   A_3126_TSC01_AC.Msg.WarningDoneL := FALSE;
   A_3126_TSC01_AC.Msg.WarningDoneMid := FALSE;
   A_3126_TSC01_AC.Msg.WarningDoneH := FALSE;
   A_3126_TSC01_AC.Msg.WarningDoneHH := FALSE;
   A_3126_TSC01_AC.Msg.FaultDoneLL := FALSE;
   A_3126_TSC01_AC.Msg.FaultDoneL := FALSE;
   A_3126_TSC01_AC.Msg.FaultDoneMid := FALSE;
   A_3126_TSC01_AC.Msg.FaultDoneH := FALSE;
   A_3126_TSC01_AC.Msg.FaultDoneHH := FALSE;
   A_3126_TSC01_AC.Msg.FaultDoneDev := FALSE;
   A_3126_TSC01_AC.Msg.FaultDoneAI := FALSE;
   A_3126_TSC01_AC.OutAlarmNrLog := 0;
   A_3126_TSC01_AC.Par.ParObjectNo := 27124;
   A_3126_TSC01_AC.Par.ParMsgType := 7252;
   A_3126_TSC01_AC.Par.ParHornCode := 10;
   A_3126_TSC01_AC.Par.ParLogOff := FALSE;
   A_3126_TSC01_AC.Par.ParSpare0401 := FALSE;
   A_3126_TSC01_AC.Par.ParValueByUser := FALSE;
   A_3126_TSC01_AC.Par.ParLimitsPc := TRUE;
   A_3126_TSC01_AC.Par.ParWago := FALSE;
   A_3126_TSC01_AC.Par.ParNoHornByWarning := FALSE;
   A_3126_TSC01_AC.Par.ParWarningLL := FALSE;
   A_3126_TSC01_AC.Par.ParWarningL := FALSE;
   A_3126_TSC01_AC.Par.ParWarningMid := FALSE;
   A_3126_TSC01_AC.Par.ParWarningH := FALSE;
   A_3126_TSC01_AC.Par.ParWarningHH := FALSE;
   A_3126_TSC01_AC.Par.ParPreAlarmLL := FALSE;
   A_3126_TSC01_AC.Par.ParPreAlarmL := FALSE;
   A_3126_TSC01_AC.Par.ParPreAlarmMid := FALSE;
   A_3126_TSC01_AC.Par.ParPreAlarmH := FALSE;
   A_3126_TSC01_AC.Par.ParPreAlarmHH := FALSE;
   A_3126_TSC01_AC.Par.ParUnitsByZeroDigit := L#0;
   A_3126_TSC01_AC.Par.ParUnitsByMaxDigit := L#25384;
   A_3126_TSC01_AC.Par.ParUnitsBy100Pc := L#10000;
   A_3126_TSC01_AC.Par.ParLimitLL := L#-1;
   A_3126_TSC01_AC.Par.ParLimitL := L#0;
   A_3126_TSC01_AC.Par.ParLimitH := L#5400;
   A_3126_TSC01_AC.Par.ParLimitHH := L#6000;
   A_3126_TSC01_AC.Par.ParMonTimeLL := 0;
   A_3126_TSC01_AC.Par.ParMonTimeL := 0;
   A_3126_TSC01_AC.Par.ParMonTimeMid := 0;
   A_3126_TSC01_AC.Par.ParMonTimeH := 0;
   A_3126_TSC01_AC.Par.ParMonTimeHH := 0;
   A_3126_TSC01_AC.Par.ParDelayTimeDown := 10;
   A_3126_TSC01_AC.Par.ParDelayTimeUp := 10;
   A_3126_TSC01_AC.Par.ParDelayTime := 30;
   A_3126_TSC01_AC.Par.OutMonTimeLL := 0;
   A_3126_TSC01_AC.Par.OutMonTimeL := 0;
   A_3126_TSC01_AC.Par.OutMonTimeMid := 0;
   A_3126_TSC01_AC.Par.OutMonTimeH := 0;
   A_3126_TSC01_AC.Par.OutMonTimeHH := 0;
   A_3126_TSC01_AC.Par.OutDelayTimeDown := 0;
   A_3126_TSC01_AC.Par.OutDelayTimeUp := 0;
   A_3126_TSC01_AC.Par.OutDelayTime := 0;
   A_3126_TSC01_AC.Par.Spare66 := 0;
   A_3126_TSC01_AF.StCode := 0;
   A_3126_TSC01_AF.InMonLL := FALSE;
   A_3126_TSC01_AF.InMonL := FALSE;
   A_3126_TSC01_AF.InMonMid := FALSE;
   A_3126_TSC01_AF.InMonH := FALSE;
   A_3126_TSC01_AF.InMonHH := FALSE;
   A_3126_TSC01_AF.spare0205 := FALSE;
   A_3126_TSC01_AF.InpFaultAI := FALSE;
   A_3126_TSC01_AF.InpFaultDev := FALSE;
   A_3126_TSC01_AF.InHWStop := FALSE;
   A_3126_TSC01_AF.InDPFault := FALSE;
   A_3126_TSC01_AF.InDisable := FALSE;
   A_3126_TSC01_AF.CmdFaultReset := FALSE;
   A_3126_TSC01_AF.InLocal := FALSE;
   A_3126_TSC01_AF.spare0305 := FALSE;
   A_3126_TSC01_AF.InReport := FALSE;
   A_3126_TSC01_AF.spare0307 := FALSE;
   A_3126_TSC01_AF.OutLL := FALSE;
   A_3126_TSC01_AF.OutL := FALSE;
   A_3126_TSC01_AF.OutH := FALSE;
   A_3126_TSC01_AF.OutHH := FALSE;
   A_3126_TSC01_AF.OutOverflow := FALSE;
   A_3126_TSC01_AF.spare0405 := FALSE;
   A_3126_TSC01_AF.OutFaultAI := FALSE;
   A_3126_TSC01_AF.spare0407 := FALSE;
   A_3126_TSC01_AF.StLL := FALSE;
   A_3126_TSC01_AF.StL := FALSE;
   A_3126_TSC01_AF.StMid := FALSE;
   A_3126_TSC01_AF.StH := FALSE;
   A_3126_TSC01_AF.StHH := FALSE;
   A_3126_TSC01_AF.StFaultAI := FALSE;
   A_3126_TSC01_AF.OutWarning := FALSE;
   A_3126_TSC01_AF.OutFaulted := FALSE;
   A_3126_TSC01_AF.InpValue := 0;
   A_3126_TSC01_AF.OutValuePc := 0;
   A_3126_TSC01_AF.OutValueUnits := L#0;
   A_3126_TSC01_AF.Msg.WarningDoneLL := FALSE;
   A_3126_TSC01_AF.Msg.WarningDoneL := FALSE;
   A_3126_TSC01_AF.Msg.WarningDoneMid := FALSE;
   A_3126_TSC01_AF.Msg.WarningDoneH := FALSE;
   A_3126_TSC01_AF.Msg.WarningDoneHH := FALSE;
   A_3126_TSC01_AF.Msg.FaultDoneLL := FALSE;
   A_3126_TSC01_AF.Msg.FaultDoneL := FALSE;
   A_3126_TSC01_AF.Msg.FaultDoneMid := FALSE;
   A_3126_TSC01_AF.Msg.FaultDoneH := FALSE;
   A_3126_TSC01_AF.Msg.FaultDoneHH := FALSE;
   A_3126_TSC01_AF.Msg.FaultDoneDev := FALSE;
   A_3126_TSC01_AF.Msg.FaultDoneAI := FALSE;
   A_3126_TSC01_AF.OutAlarmNrLog := 0;
   A_3126_TSC01_AF.Par.ParObjectNo := 27125;
   A_3126_TSC01_AF.Par.ParMsgType := 7252;
   A_3126_TSC01_AF.Par.ParHornCode := 10;
   A_3126_TSC01_AF.Par.ParLogOff := FALSE;
   A_3126_TSC01_AF.Par.ParSpare0401 := FALSE;
   A_3126_TSC01_AF.Par.ParValueByUser := FALSE;
   A_3126_TSC01_AF.Par.ParLimitsPc := TRUE;
   A_3126_TSC01_AF.Par.ParWago := FALSE;
   A_3126_TSC01_AF.Par.ParNoHornByWarning := FALSE;
   A_3126_TSC01_AF.Par.ParWarningLL := FALSE;
   A_3126_TSC01_AF.Par.ParWarningL := FALSE;
   A_3126_TSC01_AF.Par.ParWarningMid := FALSE;
   A_3126_TSC01_AF.Par.ParWarningH := FALSE;
   A_3126_TSC01_AF.Par.ParWarningHH := FALSE;
   A_3126_TSC01_AF.Par.ParPreAlarmLL := FALSE;
   A_3126_TSC01_AF.Par.ParPreAlarmL := FALSE;
   A_3126_TSC01_AF.Par.ParPreAlarmMid := FALSE;
   A_3126_TSC01_AF.Par.ParPreAlarmH := FALSE;
   A_3126_TSC01_AF.Par.ParPreAlarmHH := FALSE;
   A_3126_TSC01_AF.Par.ParUnitsByZeroDigit := L#0;
   A_3126_TSC01_AF.Par.ParUnitsByMaxDigit := L#16880;
   A_3126_TSC01_AF.Par.ParUnitsBy100Pc := L#10000;
   A_3126_TSC01_AF.Par.ParLimitLL := L#-1;
   A_3126_TSC01_AF.Par.ParLimitL := L#3000;
   A_3126_TSC01_AF.Par.ParLimitH := L#10000;
   A_3126_TSC01_AF.Par.ParLimitHH := L#10100;
   A_3126_TSC01_AF.Par.ParMonTimeLL := 0;
   A_3126_TSC01_AF.Par.ParMonTimeL := 0;
   A_3126_TSC01_AF.Par.ParMonTimeMid := 0;
   A_3126_TSC01_AF.Par.ParMonTimeH := 0;
   A_3126_TSC01_AF.Par.ParMonTimeHH := 0;
   A_3126_TSC01_AF.Par.ParDelayTimeDown := 10;
   A_3126_TSC01_AF.Par.ParDelayTimeUp := 10;
   A_3126_TSC01_AF.Par.ParDelayTime := 30;
   A_3126_TSC01_AF.Par.OutMonTimeLL := 0;
   A_3126_TSC01_AF.Par.OutMonTimeL := 0;
   A_3126_TSC01_AF.Par.OutMonTimeMid := 0;
   A_3126_TSC01_AF.Par.OutMonTimeH := 0;
   A_3126_TSC01_AF.Par.OutMonTimeHH := 0;
   A_3126_TSC01_AF.Par.OutDelayTimeDown := 0;
   A_3126_TSC01_AF.Par.OutDelayTimeUp := 0;
   A_3126_TSC01_AF.Par.OutDelayTime := 0;
   A_3126_TSC01_AF.Par.Spare66 := 0;
   A_3126_TSC01_AP.StCode := 0;
   A_3126_TSC01_AP.InMonLL := FALSE;
   A_3126_TSC01_AP.InMonL := FALSE;
   A_3126_TSC01_AP.InMonMid := FALSE;
   A_3126_TSC01_AP.InMonH := FALSE;
   A_3126_TSC01_AP.InMonHH := FALSE;
   A_3126_TSC01_AP.spare0205 := FALSE;
   A_3126_TSC01_AP.InpFaultAI := FALSE;
   A_3126_TSC01_AP.InpFaultDev := FALSE;
   A_3126_TSC01_AP.InHWStop := FALSE;
   A_3126_TSC01_AP.InDPFault := FALSE;
   A_3126_TSC01_AP.InDisable := FALSE;
   A_3126_TSC01_AP.CmdFaultReset := FALSE;
   A_3126_TSC01_AP.InLocal := FALSE;
   A_3126_TSC01_AP.spare0305 := FALSE;
   A_3126_TSC01_AP.InReport := FALSE;
   A_3126_TSC01_AP.spare0307 := FALSE;
   A_3126_TSC01_AP.OutLL := FALSE;
   A_3126_TSC01_AP.OutL := FALSE;
   A_3126_TSC01_AP.OutH := FALSE;
   A_3126_TSC01_AP.OutHH := FALSE;
   A_3126_TSC01_AP.OutOverflow := FALSE;
   A_3126_TSC01_AP.spare0405 := FALSE;
   A_3126_TSC01_AP.OutFaultAI := FALSE;
   A_3126_TSC01_AP.spare0407 := FALSE;
   A_3126_TSC01_AP.StLL := FALSE;
   A_3126_TSC01_AP.StL := FALSE;
   A_3126_TSC01_AP.StMid := FALSE;
   A_3126_TSC01_AP.StH := FALSE;
   A_3126_TSC01_AP.StHH := FALSE;
   A_3126_TSC01_AP.StFaultAI := FALSE;
   A_3126_TSC01_AP.OutWarning := FALSE;
   A_3126_TSC01_AP.OutFaulted := FALSE;
   A_3126_TSC01_AP.InpValue := 0;
   A_3126_TSC01_AP.OutValuePc := 0;
   A_3126_TSC01_AP.OutValueUnits := L#0;
   A_3126_TSC01_AP.Msg.WarningDoneLL := FALSE;
   A_3126_TSC01_AP.Msg.WarningDoneL := FALSE;
   A_3126_TSC01_AP.Msg.WarningDoneMid := FALSE;
   A_3126_TSC01_AP.Msg.WarningDoneH := FALSE;
   A_3126_TSC01_AP.Msg.WarningDoneHH := FALSE;
   A_3126_TSC01_AP.Msg.FaultDoneLL := FALSE;
   A_3126_TSC01_AP.Msg.FaultDoneL := FALSE;
   A_3126_TSC01_AP.Msg.FaultDoneMid := FALSE;
   A_3126_TSC01_AP.Msg.FaultDoneH := FALSE;
   A_3126_TSC01_AP.Msg.FaultDoneHH := FALSE;
   A_3126_TSC01_AP.Msg.FaultDoneDev := FALSE;
   A_3126_TSC01_AP.Msg.FaultDoneAI := FALSE;
   A_3126_TSC01_AP.OutAlarmNrLog := 0;
   A_3126_TSC01_AP.Par.ParObjectNo := 27126;
   A_3126_TSC01_AP.Par.ParMsgType := 7252;
   A_3126_TSC01_AP.Par.ParHornCode := 10;
   A_3126_TSC01_AP.Par.ParLogOff := FALSE;
   A_3126_TSC01_AP.Par.ParSpare0401 := FALSE;
   A_3126_TSC01_AP.Par.ParValueByUser := FALSE;
   A_3126_TSC01_AP.Par.ParLimitsPc := TRUE;
   A_3126_TSC01_AP.Par.ParWago := FALSE;
   A_3126_TSC01_AP.Par.ParNoHornByWarning := FALSE;
   A_3126_TSC01_AP.Par.ParWarningLL := FALSE;
   A_3126_TSC01_AP.Par.ParWarningL := FALSE;
   A_3126_TSC01_AP.Par.ParWarningMid := FALSE;
   A_3126_TSC01_AP.Par.ParWarningH := FALSE;
   A_3126_TSC01_AP.Par.ParWarningHH := FALSE;
   A_3126_TSC01_AP.Par.ParPreAlarmLL := FALSE;
   A_3126_TSC01_AP.Par.ParPreAlarmL := FALSE;
   A_3126_TSC01_AP.Par.ParPreAlarmMid := FALSE;
   A_3126_TSC01_AP.Par.ParPreAlarmH := FALSE;
   A_3126_TSC01_AP.Par.ParPreAlarmHH := FALSE;
   A_3126_TSC01_AP.Par.ParUnitsByZeroDigit := L#0;
   A_3126_TSC01_AP.Par.ParUnitsByMaxDigit := L#16384;
   A_3126_TSC01_AP.Par.ParUnitsBy100Pc := L#10000;
   A_3126_TSC01_AP.Par.ParLimitLL := L#-1;
   A_3126_TSC01_AP.Par.ParLimitL := L#0;
   A_3126_TSC01_AP.Par.ParLimitH := L#3150;
   A_3126_TSC01_AP.Par.ParLimitHH := L#3500;
   A_3126_TSC01_AP.Par.ParMonTimeLL := 0;
   A_3126_TSC01_AP.Par.ParMonTimeL := 0;
   A_3126_TSC01_AP.Par.ParMonTimeMid := 0;
   A_3126_TSC01_AP.Par.ParMonTimeH := 0;
   A_3126_TSC01_AP.Par.ParMonTimeHH := 0;
   A_3126_TSC01_AP.Par.ParDelayTimeDown := 10;
   A_3126_TSC01_AP.Par.ParDelayTimeUp := 10;
   A_3126_TSC01_AP.Par.ParDelayTime := 30;
   A_3126_TSC01_AP.Par.OutMonTimeLL := 0;
   A_3126_TSC01_AP.Par.OutMonTimeL := 0;
   A_3126_TSC01_AP.Par.OutMonTimeMid := 0;
   A_3126_TSC01_AP.Par.OutMonTimeH := 0;
   A_3126_TSC01_AP.Par.OutMonTimeHH := 0;
   A_3126_TSC01_AP.Par.OutDelayTimeDown := 0;
   A_3126_TSC01_AP.Par.OutDelayTimeUp := 0;
   A_3126_TSC01_AP.Par.OutDelayTime := 0;
   A_3126_TSC01_AP.Par.Spare66 := 0;
   A_3126_TSC01_AT.StCode := 0;
   A_3126_TSC01_AT.InMonLL := FALSE;
   A_3126_TSC01_AT.InMonL := FALSE;
   A_3126_TSC01_AT.InMonMid := FALSE;
   A_3126_TSC01_AT.InMonH := FALSE;
   A_3126_TSC01_AT.InMonHH := FALSE;
   A_3126_TSC01_AT.spare0205 := FALSE;
   A_3126_TSC01_AT.InpFaultAI := FALSE;
   A_3126_TSC01_AT.InpFaultDev := FALSE;
   A_3126_TSC01_AT.InHWStop := FALSE;
   A_3126_TSC01_AT.InDPFault := FALSE;
   A_3126_TSC01_AT.InDisable := FALSE;
   A_3126_TSC01_AT.CmdFaultReset := FALSE;
   A_3126_TSC01_AT.InLocal := FALSE;
   A_3126_TSC01_AT.spare0305 := FALSE;
   A_3126_TSC01_AT.InReport := FALSE;
   A_3126_TSC01_AT.spare0307 := FALSE;
   A_3126_TSC01_AT.OutLL := FALSE;
   A_3126_TSC01_AT.OutL := FALSE;
   A_3126_TSC01_AT.OutH := FALSE;
   A_3126_TSC01_AT.OutHH := FALSE;
   A_3126_TSC01_AT.OutOverflow := FALSE;
   A_3126_TSC01_AT.spare0405 := FALSE;
   A_3126_TSC01_AT.OutFaultAI := FALSE;
   A_3126_TSC01_AT.spare0407 := FALSE;
   A_3126_TSC01_AT.StLL := FALSE;
   A_3126_TSC01_AT.StL := FALSE;
   A_3126_TSC01_AT.StMid := FALSE;
   A_3126_TSC01_AT.StH := FALSE;
   A_3126_TSC01_AT.StHH := FALSE;
   A_3126_TSC01_AT.StFaultAI := FALSE;
   A_3126_TSC01_AT.OutWarning := FALSE;
   A_3126_TSC01_AT.OutFaulted := FALSE;
   A_3126_TSC01_AT.InpValue := 0;
   A_3126_TSC01_AT.OutValuePc := 0;
   A_3126_TSC01_AT.OutValueUnits := L#0;
   A_3126_TSC01_AT.Msg.WarningDoneLL := FALSE;
   A_3126_TSC01_AT.Msg.WarningDoneL := FALSE;
   A_3126_TSC01_AT.Msg.WarningDoneMid := FALSE;
   A_3126_TSC01_AT.Msg.WarningDoneH := FALSE;
   A_3126_TSC01_AT.Msg.WarningDoneHH := FALSE;
   A_3126_TSC01_AT.Msg.FaultDoneLL := FALSE;
   A_3126_TSC01_AT.Msg.FaultDoneL := FALSE;
   A_3126_TSC01_AT.Msg.FaultDoneMid := FALSE;
   A_3126_TSC01_AT.Msg.FaultDoneH := FALSE;
   A_3126_TSC01_AT.Msg.FaultDoneHH := FALSE;
   A_3126_TSC01_AT.Msg.FaultDoneDev := FALSE;
   A_3126_TSC01_AT.Msg.FaultDoneAI := FALSE;
   A_3126_TSC01_AT.OutAlarmNrLog := 0;
   A_3126_TSC01_AT.Par.ParObjectNo := 27127;
   A_3126_TSC01_AT.Par.ParMsgType := 7252;
   A_3126_TSC01_AT.Par.ParHornCode := 10;
   A_3126_TSC01_AT.Par.ParLogOff := FALSE;
   A_3126_TSC01_AT.Par.ParSpare0401 := FALSE;
   A_3126_TSC01_AT.Par.ParValueByUser := FALSE;
   A_3126_TSC01_AT.Par.ParLimitsPc := TRUE;
   A_3126_TSC01_AT.Par.ParWago := FALSE;
   A_3126_TSC01_AT.Par.ParNoHornByWarning := FALSE;
   A_3126_TSC01_AT.Par.ParWarningLL := FALSE;
   A_3126_TSC01_AT.Par.ParWarningL := FALSE;
   A_3126_TSC01_AT.Par.ParWarningMid := FALSE;
   A_3126_TSC01_AT.Par.ParWarningH := FALSE;
   A_3126_TSC01_AT.Par.ParWarningHH := FALSE;
   A_3126_TSC01_AT.Par.ParPreAlarmLL := FALSE;
   A_3126_TSC01_AT.Par.ParPreAlarmL := FALSE;
   A_3126_TSC01_AT.Par.ParPreAlarmMid := FALSE;
   A_3126_TSC01_AT.Par.ParPreAlarmH := FALSE;
   A_3126_TSC01_AT.Par.ParPreAlarmHH := FALSE;
   A_3126_TSC01_AT.Par.ParUnitsByZeroDigit := L#0;
   A_3126_TSC01_AT.Par.ParUnitsByMaxDigit := L#16384;
   A_3126_TSC01_AT.Par.ParUnitsBy100Pc := L#10000;
   A_3126_TSC01_AT.Par.ParLimitLL := L#-1;
   A_3126_TSC01_AT.Par.ParLimitL := L#0;
   A_3126_TSC01_AT.Par.ParLimitH := L#7000;
   A_3126_TSC01_AT.Par.ParLimitHH := L#8000;
   A_3126_TSC01_AT.Par.ParMonTimeLL := 0;
   A_3126_TSC01_AT.Par.ParMonTimeL := 0;
   A_3126_TSC01_AT.Par.ParMonTimeMid := 0;
   A_3126_TSC01_AT.Par.ParMonTimeH := 0;
   A_3126_TSC01_AT.Par.ParMonTimeHH := 0;
   A_3126_TSC01_AT.Par.ParDelayTimeDown := 10;
   A_3126_TSC01_AT.Par.ParDelayTimeUp := 10;
   A_3126_TSC01_AT.Par.ParDelayTime := 30;
   A_3126_TSC01_AT.Par.OutMonTimeLL := 0;
   A_3126_TSC01_AT.Par.OutMonTimeL := 0;
   A_3126_TSC01_AT.Par.OutMonTimeMid := 0;
   A_3126_TSC01_AT.Par.OutMonTimeH := 0;
   A_3126_TSC01_AT.Par.OutMonTimeHH := 0;
   A_3126_TSC01_AT.Par.OutDelayTimeDown := 0;
   A_3126_TSC01_AT.Par.OutDelayTimeUp := 0;
   A_3126_TSC01_AT.Par.OutDelayTime := 0;
   A_3126_TSC01_AT.Par.Spare66 := 0;
      #A_3125_TSC01_COM.Par.ParMovidrive                            :=1;
      #A_3125_TSC01_COM.Par.ParSinamics                             :=0;
      #A_3125_TSC01_COM.Par.ParMicromaster                          :=0;
      #A_3125_TSC01_COM.Par.ParABB                                  :=0;
      #A_3125_TSC01_COM.Par.ParNord                                 :=0;
      #A_3125_TSC01_COM.Par.ParDanfoss                              :=0;
      #A_3125_TSC01_COM.Par.ParIOByteNo                             :=0;
      #A_3125_TSC01_AC.Par.ParObjectNo                             :=27111;
      #A_3125_TSC01_AC.Par.ParHornCode                             :=10;
      #A_3125_TSC01_AC.Par.ParMsgType                              :=7252;
      #A_3125_TSC01_AC.Par.ParUnitsByZeroDigit                     :=L#0;
      #A_3125_TSC01_AC.Par.ParUnitsByMaxDigit                      :=L#25384;
      #A_3125_TSC01_AC.Par.ParUnitsBy100Pc                         :=L#10000;
      #A_3125_TSC01_AC.Par.ParDelayTimeDown                        :=10;
      #A_3125_TSC01_AC.Par.ParDelayTimeUp                          :=10;
      #A_3125_TSC01_AC.Par.ParDelayTime                            :=30;
      #A_3125_TSC01_AC.Par.ParLimitLL                              :=L#-1;
      #A_3125_TSC01_AC.Par.ParLimitL                               :=L#0;
      #A_3125_TSC01_AC.Par.ParLimitH                               :=L#5400;
      #A_3125_TSC01_AC.Par.ParLimitHH                              :=L#6000;
      #A_3125_TSC01_AC.Par.ParMonTimeLL                            :=0;
      #A_3125_TSC01_AC.Par.ParMonTimeL                             :=0;
      #A_3125_TSC01_AC.Par.ParMonTimeMid                           :=0;
      #A_3125_TSC01_AC.Par.ParMonTimeH                             :=0;
      #A_3125_TSC01_AC.Par.ParMonTimeHH                            :=0;
      #A_3125_TSC01_AC.Par.ParLogOff                               :=False;
      #A_3125_TSC01_AC.Par.ParValueByUser                          :=False;
      #A_3125_TSC01_AC.Par.ParLimitsPc                             :=True;
      #A_3125_TSC01_AC.Par.ParWago                                 :=False;
      #A_3125_TSC01_AC.Par.ParNoHornByWarning                      :=False;
      #A_3125_TSC01_AC.Par.ParWarningLL                            :=False;
      #A_3125_TSC01_AC.Par.ParWarningL                             :=False;
      #A_3125_TSC01_AC.Par.ParWarningMid                           :=False;
      #A_3125_TSC01_AC.Par.ParWarningH                             :=False;
      #A_3125_TSC01_AC.Par.ParWarningHH                            :=False;
      #A_3125_TSC01_AC.Par.ParPreAlarmLL                           :=False;
      #A_3125_TSC01_AC.Par.ParPreAlarmL                            :=False;
      #A_3125_TSC01_AC.Par.ParPreAlarmMid                          :=False;
      #A_3125_TSC01_AC.Par.ParPreAlarmH                            :=False;
      #A_3125_TSC01_AC.Par.ParPreAlarmHH                           :=False;
      #A_3125_TSC01_AF.Par.ParObjectNo                             :=27112;
      #A_3125_TSC01_AF.Par.ParHornCode                             :=10;
      #A_3125_TSC01_AF.Par.ParMsgType                              :=7252;
      #A_3125_TSC01_AF.Par.ParUnitsByZeroDigit                     :=L#0;
      #A_3125_TSC01_AF.Par.ParUnitsByMaxDigit                      :=L#16880;
      #A_3125_TSC01_AF.Par.ParUnitsBy100Pc                         :=L#10000;
      #A_3125_TSC01_AF.Par.ParDelayTimeDown                        :=10;
      #A_3125_TSC01_AF.Par.ParDelayTimeUp                          :=10;
      #A_3125_TSC01_AF.Par.ParDelayTime                            :=30;
      #A_3125_TSC01_AF.Par.ParLimitLL                              :=L#-1;
      #A_3125_TSC01_AF.Par.ParLimitL                               :=L#3000;
      #A_3125_TSC01_AF.Par.ParLimitH                               :=L#10000;
      #A_3125_TSC01_AF.Par.ParLimitHH                              :=L#10100;
      #A_3125_TSC01_AF.Par.ParMonTimeLL                            :=0;
      #A_3125_TSC01_AF.Par.ParMonTimeL                             :=0;
      #A_3125_TSC01_AF.Par.ParMonTimeMid                           :=0;
      #A_3125_TSC01_AF.Par.ParMonTimeH                             :=0;
      #A_3125_TSC01_AF.Par.ParMonTimeHH                            :=0;
      #A_3125_TSC01_AF.Par.ParLogOff                               :=False;
      #A_3125_TSC01_AF.Par.ParValueByUser                          :=False;
      #A_3125_TSC01_AF.Par.ParLimitsPc                             :=True;
      #A_3125_TSC01_AF.Par.ParWago                                 :=False;
      #A_3125_TSC01_AF.Par.ParNoHornByWarning                      :=False;
      #A_3125_TSC01_AF.Par.ParWarningLL                            :=False;
      #A_3125_TSC01_AF.Par.ParWarningL                             :=False;
      #A_3125_TSC01_AF.Par.ParWarningMid                           :=False;
      #A_3125_TSC01_AF.Par.ParWarningH                             :=False;
      #A_3125_TSC01_AF.Par.ParWarningHH                            :=False;
      #A_3125_TSC01_AF.Par.ParPreAlarmLL                           :=False;
      #A_3125_TSC01_AF.Par.ParPreAlarmL                            :=False;
      #A_3125_TSC01_AF.Par.ParPreAlarmMid                          :=False;
      #A_3125_TSC01_AF.Par.ParPreAlarmH                            :=False;
      #A_3125_TSC01_AF.Par.ParPreAlarmHH                           :=False;
      #A_3125_TSC01_AT.Par.ParObjectNo                             :=27113;
      #A_3125_TSC01_AT.Par.ParHornCode                             :=10;
      #A_3125_TSC01_AT.Par.ParMsgType                              :=7252;
      #A_3125_TSC01_AT.Par.ParUnitsByZeroDigit                     :=L#0;
      #A_3125_TSC01_AT.Par.ParUnitsByMaxDigit                      :=L#16384;
      #A_3125_TSC01_AT.Par.ParUnitsBy100Pc                         :=L#10000;
      #A_3125_TSC01_AT.Par.ParDelayTimeDown                        :=10;
      #A_3125_TSC01_AT.Par.ParDelayTimeUp                          :=10;
      #A_3125_TSC01_AT.Par.ParDelayTime                            :=30;
      #A_3125_TSC01_AT.Par.ParLimitLL                              :=L#-1;
      #A_3125_TSC01_AT.Par.ParLimitL                               :=L#0;
      #A_3125_TSC01_AT.Par.ParLimitH                               :=L#7000;
      #A_3125_TSC01_AT.Par.ParLimitHH                              :=L#8000;
      #A_3125_TSC01_AT.Par.ParMonTimeLL                            :=0;
      #A_3125_TSC01_AT.Par.ParMonTimeL                             :=0;
      #A_3125_TSC01_AT.Par.ParMonTimeMid                           :=0;
      #A_3125_TSC01_AT.Par.ParMonTimeH                             :=0;
      #A_3125_TSC01_AT.Par.ParMonTimeHH                            :=0;
      #A_3125_TSC01_AT.Par.ParLogOff                               :=False;
      #A_3125_TSC01_AT.Par.ParValueByUser                          :=False;
      #A_3125_TSC01_AT.Par.ParLimitsPc                             :=True;
      #A_3125_TSC01_AT.Par.ParWago                                 :=False;
      #A_3125_TSC01_AT.Par.ParNoHornByWarning                      :=False;
      #A_3125_TSC01_AT.Par.ParWarningLL                            :=False;
      #A_3125_TSC01_AT.Par.ParWarningL                             :=False;
      #A_3125_TSC01_AT.Par.ParWarningMid                           :=False;
      #A_3125_TSC01_AT.Par.ParWarningH                             :=False;
      #A_3125_TSC01_AT.Par.ParWarningHH                            :=False;
      #A_3125_TSC01_AT.Par.ParPreAlarmLL                           :=False;
      #A_3125_TSC01_AT.Par.ParPreAlarmL                            :=False;
      #A_3125_TSC01_AT.Par.ParPreAlarmMid                          :=False;
      #A_3125_TSC01_AT.Par.ParPreAlarmH                            :=False;
      #A_3125_TSC01_AT.Par.ParPreAlarmHH                           :=False;
      #A_3125_TSC01_AP.Par.ParObjectNo                             :=27114;
      #A_3125_TSC01_AP.Par.ParHornCode                             :=10;
      #A_3125_TSC01_AP.Par.ParMsgType                              :=7252;
      #A_3125_TSC01_AP.Par.ParUnitsByZeroDigit                     :=L#0;
      #A_3125_TSC01_AP.Par.ParUnitsByMaxDigit                      :=L#16384;
      #A_3125_TSC01_AP.Par.ParUnitsBy100Pc                         :=L#10000;
      #A_3125_TSC01_AP.Par.ParDelayTimeDown                        :=10;
      #A_3125_TSC01_AP.Par.ParDelayTimeUp                          :=10;
      #A_3125_TSC01_AP.Par.ParDelayTime                            :=30;
      #A_3125_TSC01_AP.Par.ParLimitLL                              :=L#-1;
      #A_3125_TSC01_AP.Par.ParLimitL                               :=L#0;
      #A_3125_TSC01_AP.Par.ParLimitH                               :=L#3150;
      #A_3125_TSC01_AP.Par.ParLimitHH                              :=L#3500;
      #A_3125_TSC01_AP.Par.ParMonTimeLL                            :=0;
      #A_3125_TSC01_AP.Par.ParMonTimeL                             :=0;
      #A_3125_TSC01_AP.Par.ParMonTimeMid                           :=0;
      #A_3125_TSC01_AP.Par.ParMonTimeH                             :=0;
      #A_3125_TSC01_AP.Par.ParMonTimeHH                            :=0;
      #A_3125_TSC01_AP.Par.ParLogOff                               :=False;
      #A_3125_TSC01_AP.Par.ParValueByUser                          :=False;
      #A_3125_TSC01_AP.Par.ParLimitsPc                             :=True;
      #A_3125_TSC01_AP.Par.ParWago                                 :=False;
      #A_3125_TSC01_AP.Par.ParNoHornByWarning                      :=False;
      #A_3125_TSC01_AP.Par.ParWarningLL                            :=False;
      #A_3125_TSC01_AP.Par.ParWarningL                             :=False;
      #A_3125_TSC01_AP.Par.ParWarningMid                           :=False;
      #A_3125_TSC01_AP.Par.ParWarningH                             :=False;
      #A_3125_TSC01_AP.Par.ParWarningHH                            :=False;
      #A_3125_TSC01_AP.Par.ParPreAlarmLL                           :=False;
      #A_3125_TSC01_AP.Par.ParPreAlarmL                            :=False;
      #A_3125_TSC01_AP.Par.ParPreAlarmMid                          :=False;
      #A_3125_TSC01_AP.Par.ParPreAlarmH                            :=False;
      #A_3125_TSC01_AP.Par.ParPreAlarmHH                           :=False;
      #A_3125_TSC01.Par.ParObjectNo                             :=27107;
      #A_3125_TSC01.Par.ParMsgType                              :=7156;
      #A_3125_TSC01.Par.ParHornCode                             :=0;
      #A_3125_TSC01.Par.ParDelayChange                          :=20;
      #A_3125_TSC01.Par.ParDelayTrue                            :=10;
      #A_3125_TSC01.Par.ParDelayFalse                           :=0;
      #A_3125_TSC01.Par.ParTimeoutTrue                          :=0;
      #A_3125_TSC01.Par.ParTimeoutFalse                         :=0;
      #A_3125_TSC01.Par.ParLogOff                               :=False;
      #A_3125_TSC01.Par.Par2WorkingCond                         :=False;
      #A_3125_TSC01.Par.ParFaultRetry                           :=False;
      #A_3125_TSC01.Par.ParBinLevel                             :=False;
END_DATA_BLOCK

